// TIA Portal V17 export
// export: Created 2025-06-25T13:13:22.6426289Z, ExportSetting WithDefaults, DisplayName Totally Integrated Automation Portal, DisplayVersion V17 Update 8, DisplayName TIA Portal Openness, DisplayVersion V17 Update 8, DisplayName TIA Portal Version Control Interface, DisplayVersion V17, DisplayName STEP 7 Professional, DisplayVersion V17 Update 8, DisplayName STEP 7 Safety, DisplayVersion V17 Update 6, DisplayName WinCC Advanced, DisplayVersion V17 Update 8
FUNCTION_BLOCK "fbAlarm"   // FB40, FBD
TITLE = Alarm with time delay
{ S7_Optimized_Access := 'TRUE' }
VERSION : 0.1
// stored: AutoNumber true, IsIECCheckEnabled false, IsRetainMemResEnabled false, MemoryReserve 0, SetENOAutomatically false, UDAEnableTagReadback false
   VAR_INPUT
      bInput : Bool;
      tDelay : Time;
      bAck : Bool;
      bEnable : Bool;
   END_VAR
   VAR_OUTPUT
      bActive : Bool;
      bActiveUnack : Bool;
   END_VAR
   VAR
      DelayTimer : TON_TIME;
      Alarm : Bool;
      AlarmUnack : Bool;
      mActive : Bool;
   END_VAR
   VAR_TEMP
      DelayExpired : Bool;
   END_VAR
   VAR_TEMP   // added for the SCL form of the ladder/FBD networks
      _w1 : Bool;
   END_VAR
BEGIN

REGION Network 1: Delay: alarm must be active for a minimum time period
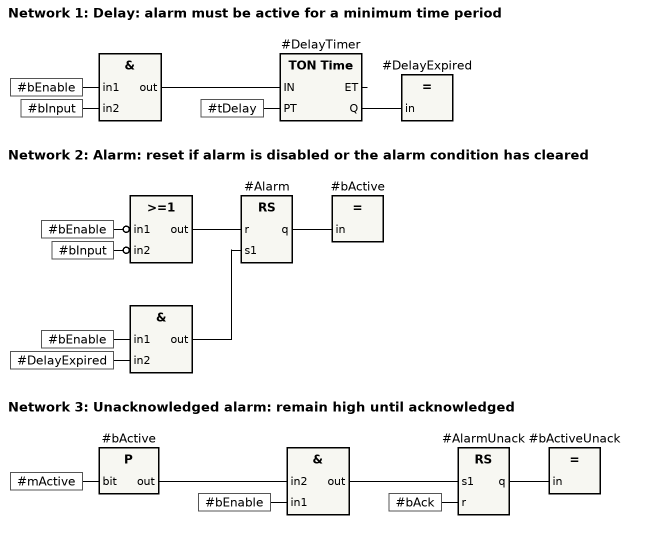
   #DelayTimer(IN := #bEnable AND #bInput, PT := #tDelay);   // TON
   #DelayExpired := #DelayTimer.Q;
END_REGION

REGION Network 2: Alarm: reset if alarm is disabled or the alarm condition has cleared
   IF NOT #bEnable OR NOT #bInput THEN
       #Alarm := FALSE;   // RS flip-flop
   END_IF;
   IF #bEnable AND #DelayExpired THEN #Alarm := TRUE; END_IF;
   #bActive := #Alarm;
END_REGION

REGION Network 3: Unacknowledged alarm: remain high until acknowledged
   #_w1 := #bActive AND NOT #mActive;   // rising edge of #bActive
   #mActive := #bActive;
   IF #bAck THEN
       #AlarmUnack := FALSE;   // RS flip-flop
   END_IF;
   IF #_w1 AND #bEnable THEN #AlarmUnack := TRUE; END_IF;
   #bActiveUnack := #AlarmUnack;
END_REGION
END_FUNCTION_BLOCK
